INTERFACE I_KinematicGroup EXTENDS I_Component, I_Override, I_TaskResult, I_Resettable

METHOD AddAcsAxis : BOOL
VAR_INPUT
	AxisId : UDINT;
END_VAR
END_METHOD

METHOD AddMcsAxis : BOOL
VAR_INPUT
	AxisId : UDINT;
END_VAR
END_METHOD

METHOD BuildGroup
VAR_INPUT
END_VAR
END_METHOD

METHOD DissolveGroup
VAR_INPUT
END_VAR
END_METHOD

{attribute 'monitoring' := 'call'}
PROPERTY Status : E_KinStatus
GET
END_GET
END_PROPERTY

END_INTERFACE

(* stored: Version 1.1.0.1, ProductVersion 3.1.4026.18
   Itf I_KinematicGroup: Id {1eeda001-fd31-4426-bdfc-22e914c643aa}
   Method AddAcsAxis: Id {3cfd2da9-2840-4f5c-b405-828b67689af0}
   Method AddMcsAxis: Id {31e282f7-0944-49e2-b9c2-8411a707a43f}
   Method BuildGroup: Id {90626a04-c63b-4c2f-a506-43293e0d366a}
   Method DissolveGroup: Id {26601a57-18ad-4890-b1fb-cfc1fe637e52}
   Property Status: Id {a64411fc-e106-43e9-9e4e-67cf0a8fc806}
   Get Get: Id {f0e908cd-d368-4bf7-b6e1-645d9ebc89ee} *)
